(* CODESYS project zadanie 1 sprawko 4.project

Project tree, tasks and I/O mapping:
  Device : CODESYS Control Win V3, CODESYS, version 3.5.20.30
    application Application
      libraries: Standard, 3.5.18.0 (System)
      task VISU_TASK (cyclic, interval 100 ms, priority 31) calls VisuElems.Visu_Prg
      task MainTask (cyclic, interval t#20ms, priority 1) calls PLC_PRG_GK
      visualisation Visualization
      program PLC_PRG_GK [LD]
  libraries: Standard, 3.5.18.0 (System); VisuElemBase, * (System)
  text list GlobalTextList
*)

// Device/Application/PLC_PRG_GK
PROGRAM PLC_PRG_GK
VAR
    S1_GK, S2_GK, S3_GK: BOOL;
    S1_mono_GK, S1_bi_GK, S2_mono_GK, S2_bi_GK, S3_mono_GK, S3_bi_GK: BOOL;
    H1_GK, H2_GK, H3_GK: BOOL;
    H4_GK, H5_GK, H6_GK: BOOL;
 	M1_GK, M2_GK, M3_GK: BOOL;
    M4_GK, M5_GK, M6_GK: BOOL;
	S2_nacisniecia_GK: WORD :=3;
	S2_impuls_GK: TIME := T#5S;
	S3_impuls_GK: TIME := T#8S;

instancjaRS: RS;
	TP_GK: TP;
	F_TRIG_0: F_TRIG;
	CTU_GK: CTU;
	TPP_GK: TP;
END_VAR

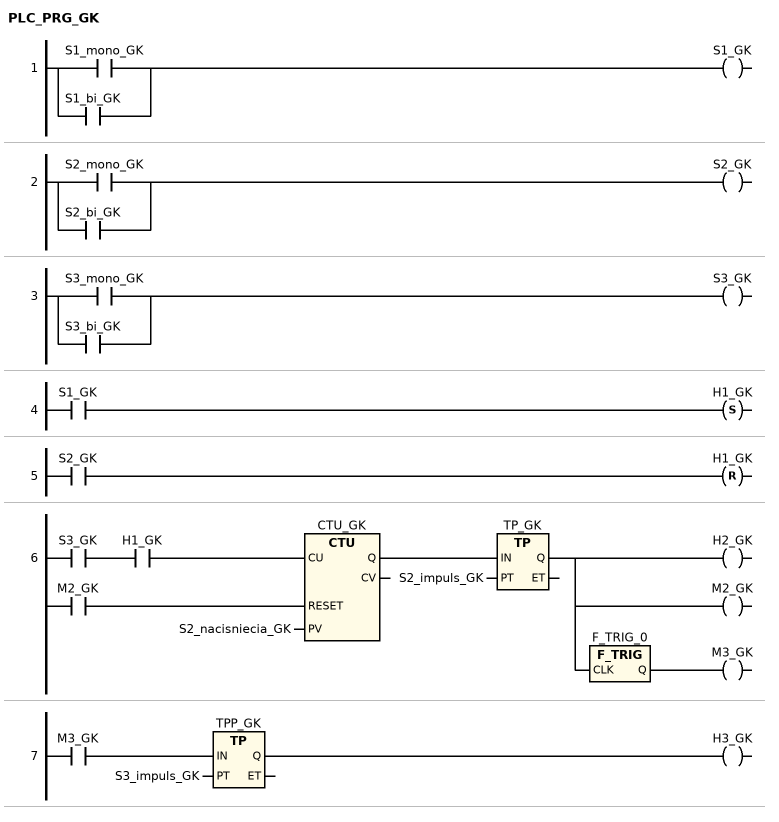
// NETWORK 1
S1_GK := S1_mono_GK OR S1_bi_GK;

// NETWORK 2
S2_GK := S2_mono_GK OR S2_bi_GK;

// NETWORK 3
S3_GK := S3_mono_GK OR S3_bi_GK;

// NETWORK 4
H1_GK S= S1_GK;

// NETWORK 5
H1_GK R= S2_GK;

// NETWORK 6
CTU_GK(CU := S3_GK AND H1_GK, RESET := M2_GK, PV := S2_nacisniecia_GK); // CTU
TP_GK(IN := CTU_GK.Q, PT := S2_impuls_GK); // TP
H2_GK := TP_GK.Q;
M2_GK := TP_GK.Q;
F_TRIG_0(CLK := TP_GK.Q); // F_TRIG
M3_GK := F_TRIG_0.Q;

// NETWORK 7
TPP_GK(IN := M3_GK, PT := S3_impuls_GK); // TP
H3_GK := TPP_GK.Q;

END_PROGRAM

// Device/Application/Visualization
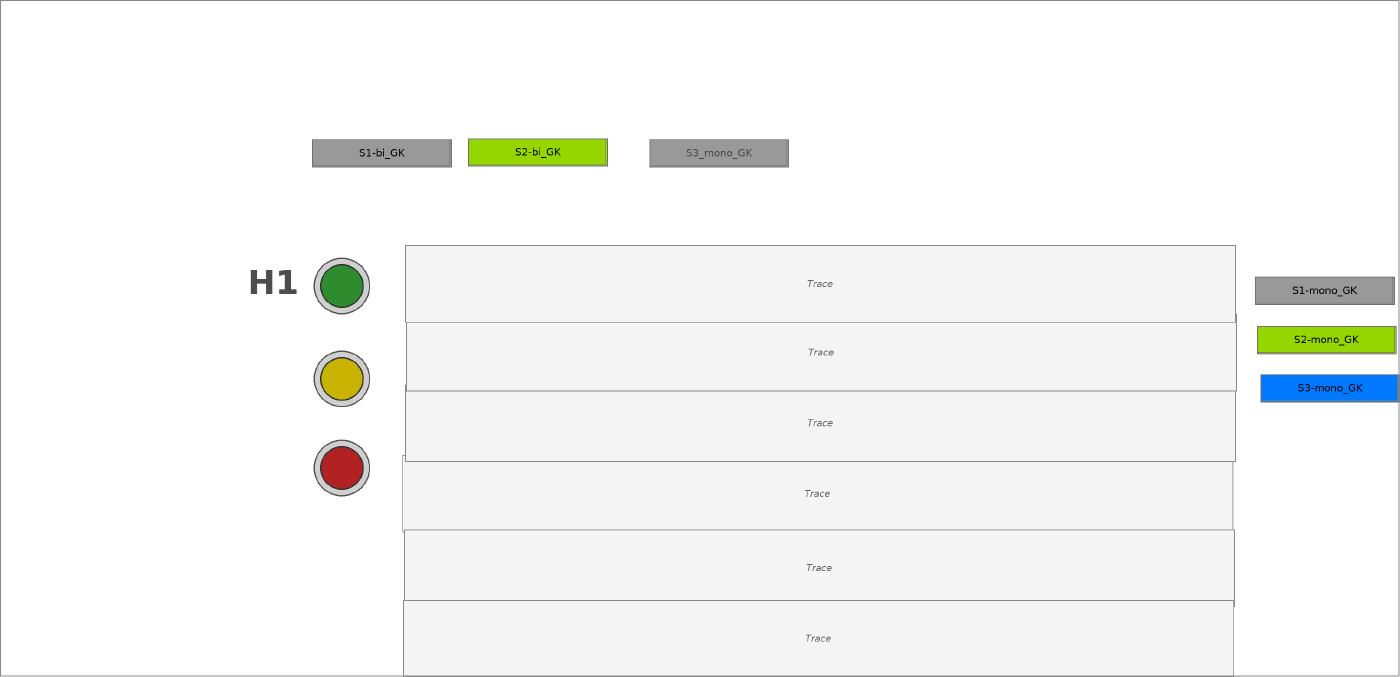
VISUALIZATION Visualization  // 1507x729
    Lamp1 (333,273 70x70), variable: PLC_PRG_GK.H1_GK, style: Lamp-Lamp1-Green
    Lamp1 (333,373 70x70), variable: PLC_PRG_GK.H2_GK, style: Lamp-Lamp1-Yellow
    Lamp1 (333,469 70x70), variable: PLC_PRG_GK.H3_GK, style: Lamp-Lamp1-Red
    Button (1351,298 150x30), "S1-mono_GK"
        tap PLC_PRG_GK.S1_mono_GK
    Button (1353,351 150x30), "S2-mono_GK"
        tap PLC_PRG_GK.S2_mono_GK
    Button (336,150 150x30), "S1-bi_GK"
        toggle PLC_PRG_GK.S1_bi_GK
    Button (504,149 150x30), "S2-bi_GK"
        toggle PLC_PRG_GK.S2_bi_GK
    Button (1357,403 150x30), "S3-mono_GK"
        tap PLC_PRG_GK.S3_mono_GK
    Button (699,150 150x30), "S3_mono_GK"
        toggle PLC_PRG_GK.S3_bi_GK
    Label (219,289 150x30), "H1"
    Trace (433,490 894x83)
    Trace (435,570 894x83)
    Trace (436,414 894x83)
    Trace (437,338 894x83)
    Trace (436,264 894x83)
    Trace (434,646 894x83)
END_VISUALIZATION
